// TIA Portal V20 export
FUNCTION_BLOCK "LER_DataTransfer"   // FB17, LAD
// stored: Access Published, MemoryReserve 100, SetENOAutomatically false
   VAR_INPUT
      LoadingCondition { ExternalAccessible := 'False'; ExternalVisible := 'False'; ExternalWritable := 'False'} : Bool;
      UnloadingCondition { ExternalAccessible := 'False'; ExternalVisible := 'False'; ExternalWritable := 'False'} : Bool;
      retryCondition : Bool := true;   // 데이터가 다음 구역으로의 이동을 확인한 신호.
   END_VAR
   VAR_OUTPUT
      loadingDataTransferDone : Bool;
      unloadingDataTransferDone : Bool;
   END_VAR
   VAR_IN_OUT
      partData1 : "LER_typePartData";
      partData2 : "LER_typePartData";
   END_VAR
   VAR
      tempActuatorLoadingActive { ExternalAccessible := 'False'; ExternalVisible := 'False'; ExternalWritable := 'False'} : Bool;
      tempActuatorUnloadingActive { ExternalAccessible := 'False'; ExternalVisible := 'False'; ExternalWritable := 'False'} : Bool;
      statRetry : Bool;   // 데이터가 다음 구역으로 이동 되기 전, 데이터가 삭제 되지 않도록 방지 하기 위한 신호.
   END_VAR
   VAR_TEMP
      tempActuatorLoadingPositiveEdge : Bool;
      tempActuatorUnloadingPositiveEdge : Bool;
      tempDeleteData : "LER_typePartData";
   END_VAR
BEGIN

REGION Network 1: Workpiece transfer positive edge
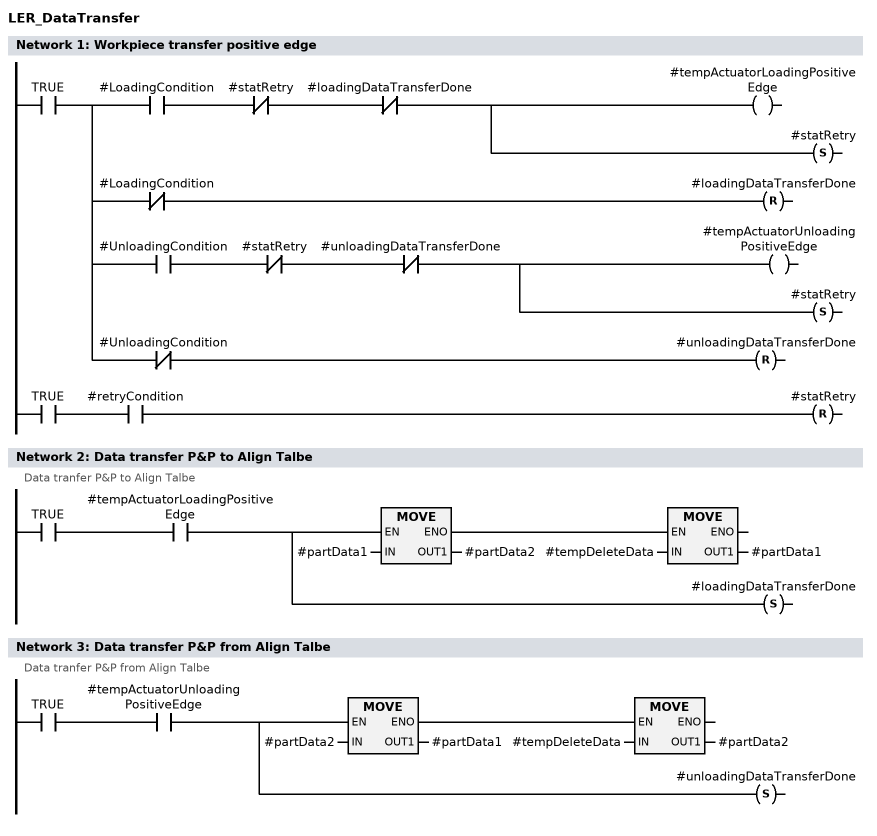
   RUNG wire#powerrail
      Contact( TRUE )
      wire#w1
      Contact( #LoadingCondition )
      I_Contact( #statRetry )
      I_Contact( #loadingDataTransferDone )
      wire#w2
      Coil( #tempActuatorLoadingPositiveEdge )
   END_RUNG
   RUNG wire#w2
      S_Coil( #statRetry )
   END_RUNG
   RUNG wire#w1
      I_Contact( #LoadingCondition )
      R_Coil( #loadingDataTransferDone )
   END_RUNG
   RUNG wire#w1
      Contact( #UnloadingCondition )
      I_Contact( #statRetry )
      I_Contact( #unloadingDataTransferDone )
      wire#w3
      Coil( #tempActuatorUnloadingPositiveEdge )
   END_RUNG
   RUNG wire#w3
      S_Coil( #statRetry )
   END_RUNG
   RUNG wire#w1
      I_Contact( #UnloadingCondition )
      R_Coil( #unloadingDataTransferDone )
   END_RUNG
   RUNG wire#powerrail
      Contact( TRUE )
      Contact( #retryCondition )
      R_Coil( #statRetry )
   END_RUNG
   // the same network as SCL:
   #tempActuatorLoadingPositiveEdge := TRUE AND #LoadingCondition AND NOT #statRetry AND NOT #loadingDataTransferDone;
   IF #tempActuatorLoadingPositiveEdge THEN #statRetry := TRUE; END_IF;
   IF TRUE AND NOT #LoadingCondition THEN #loadingDataTransferDone := FALSE; END_IF;
   #tempActuatorUnloadingPositiveEdge := TRUE AND #UnloadingCondition AND NOT #statRetry AND NOT #unloadingDataTransferDone;
   IF #tempActuatorUnloadingPositiveEdge THEN #statRetry := TRUE; END_IF;
   IF TRUE AND NOT #UnloadingCondition THEN #unloadingDataTransferDone := FALSE; END_IF;
   IF TRUE AND #retryCondition THEN #statRetry := FALSE; END_IF;
END_REGION

REGION Network 2: Data transfer P&P to Align Talbe
   // Data tranfer P&P to Align Talbe
   RUNG wire#powerrail
      Contact( TRUE )
      Contact( #tempActuatorLoadingPositiveEdge )
      wire#w1
      Move(in := #partData1, out1 => #partData2)
      Move(in := #tempDeleteData, out1 => #partData1)
   END_RUNG
   RUNG wire#w1
      S_Coil( #loadingDataTransferDone )
   END_RUNG
   // the same network as SCL:
   IF TRUE AND #tempActuatorLoadingPositiveEdge THEN
       #partData2 := #partData1;
       #partData1 := #tempDeleteData;
       #loadingDataTransferDone := TRUE;
   END_IF;
END_REGION

REGION Network 3: Data transfer P&P from Align Talbe
   // Data tranfer P&P from Align Talbe
   RUNG wire#powerrail
      Contact( TRUE )
      Contact( #tempActuatorUnloadingPositiveEdge )
      wire#w1
      Move(in := #partData2, out1 => #partData1)
      Move(in := #tempDeleteData, out1 => #partData2)
   END_RUNG
   RUNG wire#w1
      S_Coil( #unloadingDataTransferDone )
   END_RUNG
   // the same network as SCL:
   IF TRUE AND #tempActuatorUnloadingPositiveEdge THEN
       #partData1 := #partData2;
       #partData2 := #tempDeleteData;
       #unloadingDataTransferDone := TRUE;
   END_IF;
END_REGION
END_FUNCTION_BLOCK
